{attribute 'reflection'} 
{attribute 'no_explicit_call' := 'do not call this POU directly'} 
FUNCTION_BLOCK FB_ZYLINDER_TWO_WAY_MID_POS IMPLEMENTS I_PNEU_ACTOR
VAR_INPUT
END_VAR
VAR_OUTPUT
END_VAR
VAR
	{attribute 'instance-path'} 
    {attribute 'noinit'} 
	strInstancePath: STRING;
	strFullObjectPath: STRING;
	stEvent: ST_EVENT;
	bAck: BOOL;
	itfOpMode:			I_OP_MODE;
	itfValveToBase:		I_BASE_VALVE;
	itfValveToWork: 	I_BASE_VALVE;
	itfSensorInBase: 	I_BINARY_SWITCH;
	itfSensorInWork: 	I_BINARY_SWITCH;
	itfSensorInMid: 	I_BINARY_SWITCH;
	tDebounceTimeMid: TIME;
	tonDebounceTimeMid:		Tc2_Standard.TON;
	tonToBase: Tc2_Standard.TON;
	tToBase: TIME;
	tonToWork: Tc2_Standard.TON;
	tToWork: TIME;
	bViewToBase: BOOL;
	bViewToWork: BOOL;
		//Locking
	bLockWorkMovement: BOOL:=FALSE;
	bLockBaseMovement: BOOL:=FALSE;
	bLockWorkActive: BOOL:=FALSE;
	bLockBaseActive: BOOL:=FALSE;
	strLockedByObject: STRING;
	
END_VAR

METHOD FB_init : BOOL
VAR_INPUT
	bInitRetains : BOOL; // if TRUE, the retain variables are initialized (warm start / cold start)
	bInCopyCode : BOOL;  // if TRUE, the instance afterwards gets moved into the copy code (online change)
	itfOpMode:		I_OP_MODE;
	itfValveToBase: I_BASE_VALVE;
	itfValveToWork: I_BASE_VALVE;
	itfSensorInBase: I_BINARY_SWITCH;
	itfSensorInWork: I_BINARY_SWITCH;
	itfSensorInMid: I_BINARY_SWITCH;
	tTimeOutToBase: TIME;
	tTimeOutToWork: TIME;
	tDebounceTimeMid: TIME;
END_VAR
THIS^.itfOpMode:=		itfOpMode;		
THIS^.itfValveToBase:=  itfValveToBase; 
THIS^.itfValveToWork:=  itfValveToWork; 
THIS^.itfSensorInBase:= itfSensorInBase;
THIS^.itfSensorInWork:= itfSensorInWork;
THIS^.itfSensorInMid:=	itfSensorInMid;
THIS^.tToBase:= 		tTimeOutToBase;
THIS^.tToWork:= 		tTimeOutToWork;
THIS^.tDebounceTimeMid:=tDebounceTimeMid;
END_METHOD

{warning 'Methodenimplementierung hinzufügen'}
METHOD M_LockMovment
VAR_INPUT
	bLockBaseMovement	: BOOL;
	bLockWorkMovement	: BOOL;
	itfObject	: I_GENERAL_OBJECT;
END_VAR
THIS^.bLockBaseMovement:=	bLockBaseMovement;
THIS^.bLockWorkMovement:= 	bLockWorkMovement;
THIS^.strLockedByObject:= 	itfObject.P_FullObjectPath;
END_METHOD

METHOD M_Run
VAR

END_VAR
//Abarbeiten der geerbten Objekte
F_HandleInheritanceObjectInMRun(itfInheritanceObject:=THIS^.itfValveToBase,itfThisObject:=THIS^);
F_HandleInheritanceObjectInMRun(itfInheritanceObject:=THIS^.itfValveToWork,itfThisObject:=THIS^);
F_HandleInheritanceObjectInMRun(itfInheritanceObject:=THIS^.itfSensorInBase,itfThisObject:=THIS^);
F_HandleInheritanceObjectInMRun(itfInheritanceObject:=THIS^.itfSensorInWork,itfThisObject:=THIS^);
F_HandleInheritanceObjectInMRun(itfInheritanceObject:=THIS^.itfSensorInMid,itfThisObject:=THIS^);




//Handle Timeout Fault
IF tonToBase.Q AND NOT stEvent.bEventActive AND (THIS^.itfOpMode.P_OP_MODE_STATE=OP_MODE.AUTO OR THIS^.itfOpMode.P_OP_MODE_STATE=OP_MODE.DEBUG OR THIS^.itfOpMode.P_OP_MODE_STATE=OP_MODE.INIT) THEN
	stEvent.bEventActive:= TRUE;
	stEvent.enumEventType:= ENUM_EVENT_TYPE.Bl2_Message;
	stEvent.strEventText:= F_RET_TXTLIST_ENTRY(strPortNr:='851',strID:='2',strTxtLstName:='TXT_LIST_PNEMATIC_ACTOR');
	stEvent.strObject:= THIS^.P_FullObjectPath;
END_IF

IF tonToWork.Q  AND NOT stEvent.bEventActive AND (THIS^.itfOpMode.P_OP_MODE_STATE=OP_MODE.AUTO OR THIS^.itfOpMode.P_OP_MODE_STATE=OP_MODE.DEBUG OR THIS^.itfOpMode.P_OP_MODE_STATE=OP_MODE.INIT) THEN
	stEvent.bEventActive:= TRUE;
	stEvent.enumEventType:= ENUM_EVENT_TYPE.Ye4_Stateinfo;
	stEvent.strEventText:= F_RET_TXTLIST_ENTRY(strPortNr:='851',strID:='1',strTxtLstName:='TXT_LIST_PNEMATIC_ACTOR');
	stEvent.strObject:= THIS^.P_FullObjectPath;
END_IF

//Event movment is locked
IF THIS^.bLockWorkActive OR THIS^.bLockBaseActive THEN
	stEvent.bEventActive:= TRUE;
	stEvent.enumEventType:= ENUM_EVENT_TYPE.Ye4_Stateinfo;
	stEvent.strEventText:= F_RET_TXTLIST_ENTRY(strPortNr:='851',strID:='16',strTxtLstName:='TXT_LIST_PNEMATIC_ACTOR');
	stEvent.strEventText:= Tc2_Standard.CONCAT(stEvent.strEventText,' ');
	stEvent.strEventText:= Tc2_Standard.CONCAT(stEvent.strEventText,THIS^.strLockedByObject);
	stEvent.strObject:= THIS^.P_FullObjectPath;
END_IF

IF THIS^.P_Global_Ack (*AND (tonToBase.Q OR tonToWork.Q) *)THEN
	stEvent.bEventActive:= FALSE;
	tonToBase.IN:= FALSE;
	tonToWork.IN:= FALSE;
	THIS^.bLockWorkActive:=FALSE;
	THIS^.bLockBaseActive:=FALSE;
END_IF



IF THIS^.P_State=E_POS_STATE.InBasePos OR P_State=E_POS_STATE.InMidPos THEN
	tonToBase.IN:= FALSE;
END_IF
IF THIS^.P_State=E_POS_STATE.InWorkPos OR P_State=E_POS_STATE.InMidPos THEN
	tonTowork.IN:= FALSE;
END_IF

tonToWork(PT:=tToWork);
tonToBase(PT:=tToBase);

tonDebounceTimeMid.IN:=THIS^.itfSensorInMid.P_Active;
tonDebounceTimeMid(PT:=tDebounceTimeMid);
END_METHOD

{warning 'Methodenimplementierung hinzufügen'}
METHOD M_Stop
IF NOT THIS^.stEvent.bEventActive AND 
(THIS^.itfOpMode.P_OP_MODE_STATE=OP_MODE.AUTO 
OR THIS^.itfOpMode.P_OP_MODE_STATE=OP_MODE.INIT 
OR THIS^.itfOpMode.P_OP_MODE_STATE=OP_MODE.DEBUG
OR THIS^.itfOpMode.P_OP_MODE_STATE=OP_MODE.MANUAL)THEN
	THIS^.itfValveToBase.M_close();
	THIS^.itfValveToWork.M_Close();
	THIS^.tonToBase.IN:= FALSE;
	THIS^.tonToWork.IN:= FALSE;
END_IF
bViewToBase:= FALSE;
bViewToWork:= FALSE;
END_METHOD

{warning 'Methodenimplementierung hinzufügen'}
METHOD M_ToBasePos
IF NOT THIS^.stEvent.bEventActive
AND (THIS^.itfOpMode.P_OP_MODE_STATE=OP_MODE.AUTO 
OR THIS^.itfOpMode.P_OP_MODE_STATE=OP_MODE.INIT 
OR THIS^.itfOpMode.P_OP_MODE_STATE=OP_MODE.DEBUG
OR THIS^.itfOpMode.P_OP_MODE_STATE=OP_MODE.MANUAL) THEN
	IF NOT THIS^.bLockBaseMovement THEN
		THIS^.itfValveToBase.M_OPEN();
		THIS^.itfValveToWork.M_Close();
		THIS^.tonToBase.IN:= TRUE;
		THIS^.tonToWork.IN:= FALSE;
	ELSE
		THIS^.bLockBaseActive:=TRUE;
	END_IF
END_IF;

bViewToBase:= TRUE;
bViewToWork:= FALSE;
END_METHOD

{warning 'Methodenimplementierung hinzufügen'}
METHOD M_ToWorkPos
IF NOT THIS^.stEvent.bEventActive AND 
(THIS^.itfOpMode.P_OP_MODE_STATE=OP_MODE.AUTO 
OR THIS^.itfOpMode.P_OP_MODE_STATE=OP_MODE.INIT 
OR THIS^.itfOpMode.P_OP_MODE_STATE=OP_MODE.DEBUG
OR THIS^.itfOpMode.P_OP_MODE_STATE=OP_MODE.MANUAL)THEN
	IF NOT THIS^.bLockWorkMovement THEN
		THIS^.itfValveToWork.M_OPEN();
		THIS^.itfValveToBase.M_Close();
		THIS^.tonToWork.IN:= TRUE;
		THIS^.tonToBase.IN:= FALSE;
	ELSE
		THIS^.bLockWorkActive:=TRUE;
	END_IF	
END_IF
bViewToBase:= FALSE;
bViewToWork:= TRUE;
END_METHOD

{warning 'Methodenimplementierung hinzufügen'}
METHOD M_UnLockMovment
THIS^.bLockBaseMovement:=	FALSE;
THIS^.bLockWorkMovement:= 	false;
END_METHOD


PROPERTY P_Event : ST_EVENT
GET
VAR
	stEventTemp: ST_EVENT;
END_VAR
P_Event:= stEvent;
END_GET
SET
END_SET
END_PROPERTY


PROPERTY P_FullObjectPath : STRING
GET
P_FullObjectPath:= THIS^.strFullObjectPath;
END_GET
SET
THIS^.strFullObjectPath:= P_FullObjectPath;
END_SET
END_PROPERTY


PROPERTY P_Global_Ack : BOOL
GET
P_Global_Ack:= THIS^.bAck;
END_GET
SET
THIS^.bAck:=P_Global_Ack;
END_SET
END_PROPERTY


PROPERTY P_GlobalID : STRING
GET
P_GlobalID:= THIS^.strInstancePath;
END_GET
END_PROPERTY


PROPERTY P_State : E_POS_STATE
GET
P_State:=E_POS_STATE.NoDefPos;

//Actor in BasePos
IF THIS^.itfSensorInBase.P_Active THEN
	P_State:=E_POS_STATE.InBasePos;
ELSE;
END_IF

//Actor in WorkPos
IF THIS^.itfSensorInWork.P_Active THEN
	P_State:=E_POS_STATE.InWorkPos;
ELSE;
END_IF

//Actor in MidPos
IF THIS^.tonDebounceTimeMid.Q THEN
	P_State:=E_POS_STATE.InMidPos;
ELSE;
END_IF

//Actor in BasePos
IF THIS^.itfSensorInBase.P_Active AND THIS^.itfValveToBase.P_IS_OPEN THEN
	P_State:=E_POS_STATE.InBasePos;
ELSE;
END_IF

//Actor in WorkPos
IF THIS^.itfSensorInWork.P_Active AND THIS^.itfValveToWork.P_IS_OPEN THEN
	P_State:=E_POS_STATE.InWorkPos;
ELSE;
END_IF

IF  NOT THIS^.itfSensorInWork.P_Active AND NOT THIS^.itfSensorInBase.P_Active AND NOT THIS^.tonDebounceTimeMid.Q THEN
	P_State:=E_POS_STATE.NoDefPos;
	//Actor Move to Base
	IF THIS^.itfValveToBase.P_IS_OPEN AND THIS^.itfValveToWork.P_IS_CLOSE THEN
		P_State:= E_POS_STATE.MoveToBase;
	ELSE;	
	END_IF
	//Actor Move to Work
	IF THIS^.itfValveToWork.P_IS_OPEN AND THIS^.itfValveToBase.P_IS_CLOSE THEN
		P_State:= E_POS_STATE.MoveToWork;
	ELSE;	
	END_IF	
ELSE;
END_IF
IF  THIS^.itfSensorInWork.P_Active AND THIS^.itfSensorInBase.P_Active THEN
	P_State:=E_POS_STATE.NoDefPos;
END_IF

IF THIS^.bLockBaseActive THEN
	P_State:=E_POS_STATE.MoveToBaseLock;
END_IF

IF THIS^.bLockWorkActive THEN
	P_State:=E_POS_STATE.MoveToWorkLock;
END_IF
END_GET
END_PROPERTY


PROPERTY P_TimeOutToBase : TIME
GET
P_TimeOutToBase:= tonToBase.PT;
END_GET
SET
tToBase:= P_TimeOutToBase;
END_SET
END_PROPERTY


PROPERTY P_TimeOutToWork : TIME
GET
P_TimeOutToWork:= tonToWork.PT;
END_GET
SET
tToWork:= P_TimeOutToWork;
END_SET
END_PROPERTY

END_FUNCTION_BLOCK

(* stored: Version 1.1.0.1, ProductVersion 3.1.4024.12
   POU FB_ZYLINDER_TWO_WAY_MID_POS: Id {09e63394-69b6-476a-b9cf-8b051b7d25de}, SpecialFunc None
   Method FB_init: Id {71329e1a-473f-49a9-a0b1-1ea0e8bfa0d6}
   Method M_LockMovment: Id {108a1363-c87f-4147-9de7-994413c4b601}
   Method M_Run: Id {47f5c591-acd9-4d91-974b-35fead665870}
   Method M_Stop: Id {0678449c-8f91-4a98-946c-79c483d67302}
   Method M_ToBasePos: Id {e87bbd41-4857-416e-85df-bf8870f12d7f}
   Method M_ToWorkPos: Id {b114311b-1775-4bbd-80dd-eb37cae749b2}
   Method M_UnLockMovment: Id {f7a681d1-660a-421c-b333-3939992abc4f}
   Property P_Event: Id {08806105-9ae7-41f2-9a2a-c427b1ace046}
   Get Get: Id {385b2df7-b9f6-454e-a298-125c622f0f1a}
   Set Set: Id {95440580-9a3f-4b42-be8f-33e2b3a6773e}
   Property P_FullObjectPath: Id {d9abf308-6688-43fa-9197-34a77143d1f4}
   Get Get: Id {342032d3-55fd-4cbe-bc99-142e03900ba1}
   Set Set: Id {5009cca2-8850-4128-9290-b3e487193323}
   Property P_Global_Ack: Id {29116e84-5680-4460-83ac-ab6c5845b01a}
   Get Get: Id {f1185a99-68bf-48aa-8a8b-147a95aaa8f1}
   Set Set: Id {acc772a2-93d9-4600-901d-1ea5dbf9c30a}
   Property P_GlobalID: Id {f534be7c-cf76-4b12-b742-a34b42b4438a}
   Get Get: Id {b6f094a9-b949-4e67-95c8-086b8ccfa652}
   Property P_State: Id {40361d42-c67c-4373-9551-b34b28f60f94}
   Get Get: Id {4e0d1f44-2623-4e2c-921d-761ca662d624}
   Property P_TimeOutToBase: Id {0990943d-40da-4577-80cd-950feafd8cb0}
   Get Get: Id {25fe16d5-51ef-4c36-ad9b-3d30c0facc83}
   Set Set: Id {c4582022-d2f3-4469-b79d-f7e175ff308d}
   Property P_TimeOutToWork: Id {fcfee786-330d-450a-88c9-044a2452cf88}
   Get Get: Id {75de806a-6407-4d5f-b6a2-af9136f89410}
   Set Set: Id {d5161d3d-491f-4e9a-b120-87d98423a940} *)
